PROGRAM MAIN
VAR
	fbKL6581			: FB_KL6581;
	fbRec_RPS_Switch	: FB_Rec_RPS_Switch;
	dwId				: DWORD := 05057;
	stEnOceanSwitch		: STR_EnOceanSwitch;
	bReady				: BOOL;
	bBusy				: BOOL;
	bError				: BOOL;
	iErrorId			: INT;
	nidX : USINT := 1;
END_VAR

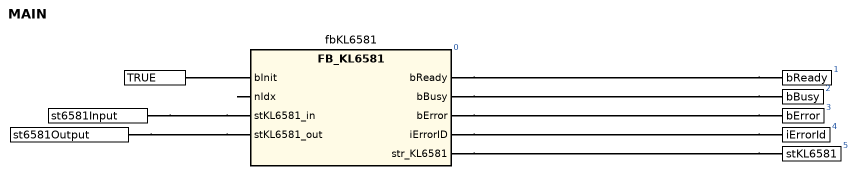
fbKL6581(bInit := TRUE, stKL6581_in := st6581Input, stKL6581_out := st6581Output); // FB_KL6581
bReady := fbKL6581.bReady;
bBusy := fbKL6581.bBusy;
bError := fbKL6581.bError;
iErrorId := fbKL6581.iErrorID;
stKL6581 := fbKL6581.str_KL6581;

END_PROGRAM

(* stored: Version 1.1.0.1, ProductVersion 3.1.4022.10
   POU MAIN: Id {cceb23df-986e-430f-9730-46b2f725b7ad}, SpecialFunc None *)
